Staubli VAL3: RobotPolish.dtx

bool bBIO[32]
  [16] = true
  [18] = true
  [22] = true
bool bDebug_PC[6] = true
bool bExit = true
bool bForceError
bool bHome
bool bInterVal
bool bIsAlarm
bool bIsPower = true
bool bJntOrPtSpd
bool bOverRun
bool bPause
bool bRefreshMsg[6]
  [0] = true
  [1] = true
  [2] = true
  [3] = true
  [4] = true
  [5] = true
bool bSuspend = true
bool bTableAlm
bool bTxtLoad
bool bUpload
bool bZero
frame fFrame = {x=1612.970915, y=39.891118, z=-82.912831, rx=0.071185, ry=-0.543234, rz=-77.228709, fatherId=world[0]}
jointRx jCurrentJoint = {j1=8.22, j2=20.1, j3=107.19, j4=-141.77, j5=44.38, j6=150.9}
jointRx jHome = {j1=40.634813, j2=24.616005, j3=104.715218, j4=-108.663007, j5=68.526435, j6=132.709111}
jointRx jJHome = {j1=11.40774, j2=30.671658, j3=109.333141, j4=204.624689, j5=51.130912, j6=-196.428273}
mdesc mNomSpeed = {accel=36, vel=60, decel=36, rmax=2000, tmax=100, blend=cartesian, leave=5, reach=5}
num nATIPress
num nATiPressBuff
num nFunctionIndex = -1
num nInterfaceType = 9
num nJntList
public num nLimitAti[6]
  [0] = 500
  [1] = 500
  [2] = 500
  [3] = 100
  [4] = 100
  [5] = 100
num nMoveID
num nPage
num nPauseTime = 6
num nSelect
num nTabSpeed = 5
num nTimeBuff = 6728.108
num nTxtSelseted = 3
num nVirtualKey = -1
num nWorkModeStatus
num nWorkingMode = 4
pointRx p = {x=-96.25, y=181, rx=-8.631, ry=175.438, rz=-89.108, fatherId=fFrame[0]}
pointRx pCurrent = {x=-7.439422, y=-0.703489, z=141.92314, rx=-0.008216, ry=-179.493493, rz=-59.800957, shoulder=lefty, elbow=epositive, wrist=wpositive, fatherId=fFrame[0]}
string sButtons[2]
  [0] = "Yes"
  [1] = "No"
string sErrorMsg[8]
  [0] = "UPS报错，检查工厂供电"
  [1] = "转台故障报警"
  [2] = "工具报警"
  [3] = "ATI与机器人通讯异常"
  [4] = "打磨力超出上限"
  [5] = "急停状态激活中"
string sItems[8]
  [0] = "信号"
  [1] = "生产"
  [2] = "TCP"
  [3] = "Frame"
  [4] = "Home"
  [5] = "速度"
  [7] = "退出"
string sMassage
string sPrdStatus[10]
  [0] = "Txt文件:"
  [1] = "TEST.txt"
  [2] = "生产状态:无生产"
  [3] = "运动状态:Move"
  [4] = "总路径个数:     1"
  [5] = "当前路径  :     1"
  [6] = "写入点个数:   902"
  [7] = "读取点个数:     1"
  [8] = "当前MoveID:     0"
  [9] = "瞬时速度  :  5.4 "
string sStrFileName[6]
  [0] = "1233"
  [1] = "BUFF"
  [2] = "TEST.txt"
  [3] = "speed of TCP.txt"
string sTxtLists[12]
  [0] = "1233"
  [1] = "BUFF"
  [2] = "TEST"
  [3] = "TEST.txt"
  [4] = "speed of TCP.txt"
string sTxtSelected = "TEST.txt"
tool tTTool = {x=1.417, y=48.029, z=261.326, rx=-28.407, ry=-42.029, rz=-19.448, fatherId=flange[0], ioLink=valve1}
public tool tTool = {x=350.22, y=-0.767094, z=232.538993, rx=-89.841339, ry=89.729222, rz=89.842087, fatherId=flange[0], ioLink=valve1}
trsf trFrame = {x=1460.596362, y=35.712914, z=-199.189903, rx=-0.117127, ry=-0.30554, rz=-53.750077}
